    //------------------------------------------------------------------------//
    // VERIFY  VERIFY VERIFY VERIFY VERIFY VERIFY VERIFY VERIFY VERIFY VERIFY //
    //------------------------------------------------------------------------//
    //Verify current substate.
A(;
L #_emc_water_subs;
L "dbCONST".BLK.EMC2.SUBS.CHARGE;
==I;
);
    S     #sqSequencer.STEP.ActionVerified; //Action verified

    //------------------------------------------------------------------------//
    // Action done:                                                           //
    //------------------------------------------------------------------------//
    O     #sqSequencer.STEP.ActionVerified;
    O     #smc.NO_VERIFIC;       //No verification , bypass verification code
    S     #sqSequencer.STEP.ActionFinished;






    //============================= STEP FOOTER ==============================//
    // AUTOCODE   AUTOCODE   AUTOCODE   AUTOCODE   AUTOCODE   AUTOCODE   AUTO //
    // Get Ready after action finished:                                       //
    //------------------------------------------------------------------------//
    A     #sqSequencer.STEP.ActionFinished;
    JCN   k006;

    //------------------------------------------------------------------------//
    // Reset Action finished flag, ready for next step action:                //
    //------------------------------------------------------------------------//
    R     #sqSequencer.STEP.ActionVerified;
    R     #sqSequencer.STEP.ActionFinished;

    //------------------------------------------------------------------------//
    // If ALL actions are finished:                                           //
    //------------------------------------------------------------------------//
    SET   ;
    S     #sqSequencer.STEP.Finished;
    R     #sqSequencer.STEP.Active;
    S     #sqSequencer.STEP.Done[06];

    //------------------------------------------------------------------------//
    // End Step action(s):                                                    //
    //------------------------------------------------------------------------//
    JU    k006;

//----------------------------------------------------------------------------//
// Finished Step Action(s):                                                   //
//----------------------------------------------------------------------------//
k006: NOP   0;

    A     #sqStepTimerExpired;
    S     #sqSequencer.STEP.WithError[06]; // Step error flag
    S     #sqSequencer.Error_Fault;
    R     #sqStepTimer.IN;

NETWORK
TITLE =S006:STEP-006::Begin Transition
    //------------------------------------------------------------------------//
    // Begin the transition code:                                             //
    //------------------------------------------------------------------------//
    A006: NOP   0;
    R     #sqStepTimer.IN;






    //============================= TRAN HEADER ==============================//
    // AUTOCODE   AUTOCODE   AUTOCODE   AUTOCODE   AUTOCODE   AUTOCODE   AUTO //
    // Bypass transition if manual jump:                                      //
    //------------------------------------------------------------------------//
    A     #sqSequencer.STEP.Finished;
    A     #smc.TRN_AND_JUMP;     //Manual jump is set Transition as bypassed
    JCN   COMM;              //exit

NETWORK
TITLE =S006::STEP 006:TRAN 010: Charge WFI complete?
//----------------------------------------------------------------------------//
// TRAN   TRAN   TRAN   TRAN   TRAN   TRAN   TRAN   TRAN   TRAN   TRAN   TRAN //
// TRAN   TRAN   TRAN   TRAN   TRAN   TRAN   TRAN   TRAN   TRAN   TRAN   TRAN //
//----------------------------------------------------------------------------//
// Check if charging WFI is completed.
//----------------------------------------------------------------------------//
// CONDITION   CONDITION   CONDITION   CONDITION   CONDITION   CONDITION   CO //
// CONDITION   CONDITION   CONDITION   CONDITION   CONDITION   CONDITION   CO //
//----------------------------------------------------------------------------//
A(;
L   #_emc_water_state;
L   "dbCONST".BLK.STATE.COMPLETED;
==I;
);






    //============================= TRAN FOOTER ==============================//
    // Transition jump control:                                               //
    //------------------------------------------------------------------------//
    A     #sqSequencer.STEP.JumpCtrl;
    S     #sqSequencer.STEP.Jump;
    S     #sqSequencer.STEP.jumpDone[06];

NETWORK
TITLE =S006:t010::TRANS-v: EXIT TRANSITION AND READY THE NEXT STEP
    //------------------------------------------------------------------------//
    // Check the jump flag and jump to the next step if the transition        //
    // condition is true and has set the jump flag:                           //
    //------------------------------------------------------------------------//
    A     #sqSequencer.STEP.Jump;
    JCN   x010;

    R     #sqSequencer.STEP.Jump;
    R     #sqSequencer.STEP.Finished;

    L     07;     // Load next STEPNO to jump to if transition satisfied
    T     #sqSequencer.STEP.NumberNext; //Next Step07.

    JU    COMM;              // Transition satisfied, Exit, go to next step
x010: NOP   0;






NETWORK
TITLE =S006::STEP-006:EXIT TRANSITION:
    //========================== STEP TRANSFER ===============================//
    // Jump to the common step progression code:                              //
    //------------------------------------------------------------------------//
    JU    COMM;






NETWORK
TITLE =S007: STEP-07::UO_MX_MAKE : Reset command
    //================================ STEP HEADER ===========================//
    // STEP007 STEP007 STEP007 STEP007
    // AUTOCODE   AUTOCODE   AUTOCODE   AUTOCODE   AUTOCODE   AUTOCODE   AUTO //
    // STEP007 STEP007 STEP007 STEP007
    //------------------------------------------------------------------------//
    // Reset CHARGE command.
    // Log Mx vessel weight.
    //------------------------------------------------------------------------//
S007: NOP   0;

      SET;
      R     #sqSequencer.STEP.jumpDone[07];
      A     #sqSequencer.CMD.Pause; //If paused jump
      JC    COMM;

NETWORK
TITLE =S007:STEP-07:Begin Action

      A     #sqSequencer.STEP.Finished;
      JC    A007; // Exit Action code, Jump to A007 Transition code

      //----------------------------------------------------------------------//
      // Begin step Action:                                                   //
      //----------------------------------------------------------------------//
      A     #sqSequencer.STEP.Active;
      JC    L007; // Action number loaded, Jump to L007--Step Action List

      //----------------------------------------------------------------------//
      // Load Default/Initial Step action number:                             //
      //----------------------------------------------------------------------//
      S     #sqSequencer.STEP.Active;
      S     #sqStepTimer.IN;
      L     1; //First Action, Step must contain Minimum one action
      T     #sqSequencer.STEP.ActionNumber;

//----------------------------------------------------------------------------//
// Step action list.                                                          //
// aann=mini Action step number(aa) inside main step number(nn)               //
// First Action aa00, Second action ab00, Third ac00, etc.                    //
//----------------------------------------------------------------------------//
L007: NOP   0;

      L     #sqSequencer.STEP.ActionNumber;
      JL    r007; //Wrong Action number
      JU    _007; //Action error handling
       JU    aa07; //ACTION-01


//----------------------------------------------------------------------------//
// More step action in the list can be inserted here, upto ab is tested:      //
//----------------------------------------------------------------------------//
r007: NOP   0; //Wrong action number
      S     #sqSequencer.Error_Fault;
      JU    k007; //Exit
_007: NOP   0; // Action error handling
      JU    k007; // Exit






NETWORK
TITLE =S007:: STEP-007:: : ACTION CODE
    //================================ ACT HEADER ============================//
    // ACTION ACTION ACTION ACTION ACTION ACTION ACTION ACTION ACTION ACTION  //
    // AUTOCODE   AUTOCODE   AUTOCODE   AUTOCODE   AUTOCODE   AUTOCODE   AUTO //
    // ACTION ACTION ACTION ACTION ACTION ACTION ACTION ACTION ACTION ACTION  //
    //------------------------------------------------------------------------//
    // //Reset CHARGE command.
    aa07: NOP   0;

    //------------------------------------------------------------------------//
    // ACT ACT ACT ACT ACT ACT ACT ACT ACT ACT ACT ACT ACT ACT ACT ACT ACT    //
    //------------------------------------------------------------------------//
    L "dbCONST".BLK.CMD.STOP;
T #_emv_inlet_cmd;

// Reset flag.
SET;
R #_cmd_charge;

    //------------------------------------------------------------------------//
    // VERIFY  VERIFY VERIFY VERIFY VERIFY VERIFY VERIFY VERIFY VERIFY VERIFY //
    //------------------------------------------------------------------------//
    A "uncondJump";
    S     #sqSequencer.STEP.ActionVerified; //Action verified

    //------------------------------------------------------------------------//
    // Action done:                                                           //
    //------------------------------------------------------------------------//
    O     #sqSequencer.STEP.ActionVerified;
    O     #smc.NO_VERIFIC;       //No verification , bypass verification code
    S     #sqSequencer.STEP.ActionFinished;






    //============================= STEP FOOTER ==============================//
    // AUTOCODE   AUTOCODE   AUTOCODE   AUTOCODE   AUTOCODE   AUTOCODE   AUTO //
    // Get Ready after action finished:                                       //
    //------------------------------------------------------------------------//
    A     #sqSequencer.STEP.ActionFinished;
    JCN   k007;

    //------------------------------------------------------------------------//
    // Reset Action finished flag, ready for next step action:                //
    //------------------------------------------------------------------------//
    R     #sqSequencer.STEP.ActionVerified;
    R     #sqSequencer.STEP.ActionFinished;

    //------------------------------------------------------------------------//
    // If ALL actions are finished:                                           //
    //------------------------------------------------------------------------//
    SET   ;
    S     #sqSequencer.STEP.Finished;
    R     #sqSequencer.STEP.Active;
    S     #sqSequencer.STEP.Done[07];

    //------------------------------------------------------------------------//
    // End Step action(s):                                                    //
    //------------------------------------------------------------------------//
    JU    k007;

//----------------------------------------------------------------------------//
// Finished Step Action(s):                                                   //
//----------------------------------------------------------------------------//
k007: NOP   0;

    A     #sqStepTimerExpired;
    S     #sqSequencer.STEP.WithError[07]; // Step error flag
    S     #sqSequencer.Error_Fault;
    R     #sqStepTimer.IN;

NETWORK
TITLE =S007:STEP-007::Begin Transition
    //------------------------------------------------------------------------//
    // Begin the transition code:                                             //
    //------------------------------------------------------------------------//
    A007: NOP   0;
    R     #sqStepTimer.IN;






    //============================= TRAN HEADER ==============================//
    // AUTOCODE   AUTOCODE   AUTOCODE   AUTOCODE   AUTOCODE   AUTOCODE   AUTO //
    // Bypass transition if manual jump:                                      //
    //------------------------------------------------------------------------//
    A     #sqSequencer.STEP.Finished;
    A     #smc.TRN_AND_JUMP;     //Manual jump is set Transition as bypassed
    JCN   COMM;              //exit

NETWORK
TITLE =S007::STEP 007:TRAN 011: Sprayball inlet valves closed
//----------------------------------------------------------------------------//
// TRAN   TRAN   TRAN   TRAN   TRAN   TRAN   TRAN   TRAN   TRAN   TRAN   TRAN //
// TRAN   TRAN   TRAN   TRAN   TRAN   TRAN   TRAN   TRAN   TRAN   TRAN   TRAN //
//----------------------------------------------------------------------------//
// Jump if sprayball valves closed
//----------------------------------------------------------------------------//
// CONDITION   CONDITION   CONDITION   CONDITION   CONDITION   CONDITION   CO //
// CONDITION   CONDITION   CONDITION   CONDITION   CONDITION   CONDITION   CO //
//----------------------------------------------------------------------------//
A(;
L   #_emv_inlet_state;
L   "dbCONST".BLK.STATE.STOPPED;
==I;
);






    //============================= TRAN FOOTER ==============================//
    // Transition jump control:                                               //
    //------------------------------------------------------------------------//
    A     #sqSequencer.STEP.JumpCtrl;
    S     #sqSequencer.STEP.Jump;
    S     #sqSequencer.STEP.jumpDone[07];

NETWORK
TITLE =S007:t011::TRANS-v: EXIT TRANSITION AND READY THE NEXT STEP
    //------------------------------------------------------------------------//
    // Check the jump flag and jump to the next step if the transition        //
    // condition is true and has set the jump flag:                           //
    //------------------------------------------------------------------------//
    A     #sqSequencer.STEP.Jump;
    JCN   x011;

    R     #sqSequencer.STEP.Jump;
    R     #sqSequencer.STEP.Finished;

    L     03;     // Load next STEPNO to jump to if transition satisfied
    T     #sqSequencer.STEP.NumberNext; //Next Step03.

    JU    COMM;              // Transition satisfied, Exit, go to next step
x011: NOP   0;






NETWORK
TITLE =S007::STEP-007:EXIT TRANSITION:
    //========================== STEP TRANSFER ===============================//
    // Jump to the common step progression code:                              //
    //------------------------------------------------------------------------//
    JU    COMM;






NETWORK
TITLE =S008: STEP-08::UO_MX_MAKE : MIXING vessel contents
    //================================ STEP HEADER ===========================//
    // STEP008 STEP008 STEP008 STEP008
    // AUTOCODE   AUTOCODE   AUTOCODE   AUTOCODE   AUTOCODE   AUTOCODE   AUTO //
    // STEP008 STEP008 STEP008 STEP008
    //------------------------------------------------------------------------//
    // Set ema_vessel to substate MIX with pre-selected runtime and speed.
    //------------------------------------------------------------------------//
S008: NOP   0;

      SET;
      R     #sqSequencer.STEP.jumpDone[08];
      A     #sqSequencer.CMD.Pause; //If paused jump
      JC    COMM;

NETWORK
TITLE =S008:STEP-08:Begin Action

      A     #sqSequencer.STEP.Finished;
      JC    A008; // Exit Action code, Jump to A008 Transition code

      //----------------------------------------------------------------------//
      // Begin step Action:                                                   //
      //----------------------------------------------------------------------//
      A     #sqSequencer.STEP.Active;
      JC    L008; // Action number loaded, Jump to L008--Step Action List

      //----------------------------------------------------------------------//
      // Load Default/Initial Step action number:                             //
      //----------------------------------------------------------------------//
      S     #sqSequencer.STEP.Active;
      S     #sqStepTimer.IN;
      L     1; //First Action, Step must contain Minimum one action
      T     #sqSequencer.STEP.ActionNumber;

//----------------------------------------------------------------------------//
// Step action list.                                                          //
// aann=mini Action step number(aa) inside main step number(nn)               //
// First Action aa00, Second action ab00, Third ac00, etc.                    //
//----------------------------------------------------------------------------//
L008: NOP   0;

      L     #sqSequencer.STEP.ActionNumber;
      JL    r008; //Wrong Action number
      JU    _008; //Action error handling
       JU    aa08; //ACTION-01
JU    ab08; //ACTION-02


//----------------------------------------------------------------------------//
// More step action in the list can be inserted here, upto ab is tested:      //
//----------------------------------------------------------------------------//
r008: NOP   0; //Wrong action number
      S     #sqSequencer.Error_Fault;
      JU    k008; //Exit
_008: NOP   0; // Action error handling
      JU    k008; // Exit






NETWORK
TITLE =S008:: STEP-008:: : ACTION CODE
    //================================ ACT HEADER ============================//
    // ACTION ACTION ACTION ACTION ACTION ACTION ACTION ACTION ACTION ACTION  //
    // AUTOCODE   AUTOCODE   AUTOCODE   AUTOCODE   AUTOCODE   AUTOCODE   AUTO //
    // ACTION ACTION ACTION ACTION ACTION ACTION ACTION ACTION ACTION ACTION  //
    //------------------------------------------------------------------------//
    // //Set substate to safe state and stop ema_vessel.
    aa08: NOP   0;

    //------------------------------------------------------------------------//
    // ACT ACT ACT ACT ACT ACT ACT ACT ACT ACT ACT ACT ACT ACT ACT ACT ACT    //
    //------------------------------------------------------------------------//
    L "dbCONST".BLK.CMD.STOP;
T  #_ema_vessel_cmd;

    //------------------------------------------------------------------------//
    // VERIFY  VERIFY VERIFY VERIFY VERIFY VERIFY VERIFY VERIFY VERIFY VERIFY //
    //------------------------------------------------------------------------//
    //Verify ema_vessel stopped status.
A(;
L #_ema_vessel_state;
L "dbCONST".BLK.STATE.STOPPED;
==I;
);
    S     #sqSequencer.STEP.ActionVerified; //Action verified

    //------------------------------------------------------------------------//
    // Action done:                                                           //
    //------------------------------------------------------------------------//
    O     #sqSequencer.STEP.ActionVerified;
    O     #smc.NO_VERIFIC;       //No verification , bypass verification code
    S     #sqSequencer.STEP.ActionFinished;






    //============================= ACT FOOTER ===============================//
    // AUTOCODE   AUTOCODE   AUTOCODE   AUTOCODE   AUTOCODE   AUTOCODE   AUTO //
    // Get Ready after action finished:                                       //
    //------------------------------------------------------------------------//
    A     #sqSequencer.STEP.ActionFinished;
    JCN   k008;

    //------------------------------------------------------------------------//
    // Reset Action finished flag, ready for next step action:                //
    //------------------------------------------------------------------------//
    R     #sqSequencer.STEP.ActionVerified;
    R     #sqSequencer.STEP.ActionFinished;

    //------------------------------------------------------------------------//
    // Load Next Step Action number:                                          //
    //------------------------------------------------------------------------//
    L     02; //Load next Action
    T     #sqSequencer.STEP.ActionNumber;






NETWORK
TITLE =S008:: STEP-008:: : ACTION CODE
    //================================ ACT HEADER ============================//
    // ACTION ACTION ACTION ACTION ACTION ACTION ACTION ACTION ACTION ACTION  //
    // AUTOCODE   AUTOCODE   AUTOCODE   AUTOCODE   AUTOCODE   AUTOCODE   AUTO //
    // ACTION ACTION ACTION ACTION ACTION ACTION ACTION ACTION ACTION ACTION  //
    //------------------------------------------------------------------------//
    // //Set ema_vessel to substate MIX with pre-selected timeout and speed.
    ab08: NOP   0;

    //------------------------------------------------------------------------//
    // ACT ACT ACT ACT ACT ACT ACT ACT ACT ACT ACT ACT ACT ACT ACT ACT ACT    //
    //------------------------------------------------------------------------//
    //Transfer input parameter from HMI to EM
//Load Agitator speed setpoint.
L #_fp_speed_setpoint;
T #_ema_vessel_setpoint;
//Load Agitator runtime.
L #_fp_time_make_agit;
L 1000;
*I;
T #_ema_vessel_runtime;

// Start Agitator
L "dbCONST".BLK.EMA1.SUBS.MIX;
T #_ema_vessel_subs;
L "dbCONST".BLK.CMD.START;
T #_ema_vessel_cmd;

    //------------------------------------------------------------------------//
    // VERIFY  VERIFY VERIFY VERIFY VERIFY VERIFY VERIFY VERIFY VERIFY VERIFY //
    //------------------------------------------------------------------------//
    //Substate changed to Mix.
A(;
L #_ema_vessel_subs;
L "dbCONST".BLK.EMA1.SUBS.MIX;
==I;
);
    S     #sqSequencer.STEP.ActionVerified; //Action verified

    //------------------------------------------------------------------------//
    // Action done:                                                           //
    //------------------------------------------------------------------------//
    O     #sqSequencer.STEP.ActionVerified;
    O     #smc.NO_VERIFIC;       //No verification , bypass verification code
    S     #sqSequencer.STEP.ActionFinished;






    //============================= STEP FOOTER ==============================//
    // AUTOCODE   AUTOCODE   AUTOCODE   AUTOCODE   AUTOCODE   AUTOCODE   AUTO //
    // Get Ready after action finished:                                       //
    //------------------------------------------------------------------------//
    A     #sqSequencer.STEP.ActionFinished;
    JCN   k008;

    //------------------------------------------------------------------------//
    // Reset Action finished flag, ready for next step action:                //
    //------------------------------------------------------------------------//
    R     #sqSequencer.STEP.ActionVerified;
    R     #sqSequencer.STEP.ActionFinished;

    //------------------------------------------------------------------------//
    // If ALL actions are finished:                                           //
    //------------------------------------------------------------------------//
    SET   ;
    S     #sqSequencer.STEP.Finished;
    R     #sqSequencer.STEP.Active;
    S     #sqSequencer.STEP.Done[08];

    //------------------------------------------------------------------------//
    // End Step action(s):                                                    //
    //------------------------------------------------------------------------//
    JU    k008;

//----------------------------------------------------------------------------//
// Finished Step Action(s):                                                   //
//----------------------------------------------------------------------------//
k008: NOP   0;

    A     #sqStepTimerExpired;
    S     #sqSequencer.STEP.WithError[08]; // Step error flag
    S     #sqSequencer.Error_Fault;
    R     #sqStepTimer.IN;

NETWORK
TITLE =S008:STEP-008::Begin Transition
    //------------------------------------------------------------------------//
    // Begin the transition code:                                             //
    //------------------------------------------------------------------------//
    A008: NOP   0;
    R     #sqStepTimer.IN;






    //============================= TRAN HEADER ==============================//
    // AUTOCODE   AUTOCODE   AUTOCODE   AUTOCODE   AUTOCODE   AUTOCODE   AUTO //
    // Bypass transition if manual jump:                                      //
    //------------------------------------------------------------------------//
    A     #sqSequencer.STEP.Finished;
    A     #smc.TRN_AND_JUMP;     //Manual jump is set Transition as bypassed
    JCN   COMM;              //exit

NETWORK
TITLE =S008::STEP 008:TRAN 012: Mixing complete?
//----------------------------------------------------------------------------//
// TRAN   TRAN   TRAN   TRAN   TRAN   TRAN   TRAN   TRAN   TRAN   TRAN   TRAN //
// TRAN   TRAN   TRAN   TRAN   TRAN   TRAN   TRAN   TRAN   TRAN   TRAN   TRAN //
//----------------------------------------------------------------------------//
// Check if Mixing is completed.
//----------------------------------------------------------------------------//
// CONDITION   CONDITION   CONDITION   CONDITION   CONDITION   CONDITION   CO //
// CONDITION   CONDITION   CONDITION   CONDITION   CONDITION   CONDITION   CO //
//----------------------------------------------------------------------------//
A(;
L   #_ema_vessel_state;
L   "dbCONST".BLK.STATE.COMPLETED;
==I;
);






    //============================= TRAN FOOTER ==============================//
    // Transition jump control:                                               //
    //------------------------------------------------------------------------//
    A     #sqSequencer.STEP.JumpCtrl;
    S     #sqSequencer.STEP.Jump;
    S     #sqSequencer.STEP.jumpDone[08];

NETWORK
TITLE =S008:t012::TRANS-v: EXIT TRANSITION AND READY THE NEXT STEP
    //------------------------------------------------------------------------//
    // Check the jump flag and jump to the next step if the transition        //
    // condition is true and has set the jump flag:                           //
    //------------------------------------------------------------------------//
    A     #sqSequencer.STEP.Jump;
    JCN   x012;

    R     #sqSequencer.STEP.Jump;
    R     #sqSequencer.STEP.Finished;

    L     09;     // Load next STEPNO to jump to if transition satisfied
    T     #sqSequencer.STEP.NumberNext; //Next Step09.

    JU    COMM;              // Transition satisfied, Exit, go to next step
x012: NOP   0;






NETWORK
TITLE =S008::STEP-008:EXIT TRANSITION:
    //========================== STEP TRANSFER ===============================//
    // Jump to the common step progression code:                              //
    //------------------------------------------------------------------------//
    JU    COMM;






NETWORK
TITLE =S009: STEP-09::UO_MX_MAKE : Reset MIX command.
    //================================ STEP HEADER ===========================//
    // STEP009 STEP009 STEP009 STEP009
    // AUTOCODE   AUTOCODE   AUTOCODE   AUTOCODE   AUTOCODE   AUTOCODE   AUTO //
    // STEP009 STEP009 STEP009 STEP009
    //------------------------------------------------------------------------//
    // Reset MIX command.
    //------------------------------------------------------------------------//
S009: NOP   0;

      SET;
      R     #sqSequencer.STEP.jumpDone[09];
      A     #sqSequencer.CMD.Pause; //If paused jump
      JC    COMM;

NETWORK
TITLE =S009:STEP-09:Begin Action

      A     #sqSequencer.STEP.Finished;
      JC    A009; // Exit Action code, Jump to A009 Transition code

      //----------------------------------------------------------------------//
      // Begin step Action:                                                   //
      //----------------------------------------------------------------------//
      A     #sqSequencer.STEP.Active;
      JC    L009; // Action number loaded, Jump to L009--Step Action List

      //----------------------------------------------------------------------//
      // Load Default/Initial Step action number:                             //
      //----------------------------------------------------------------------//
      S     #sqSequencer.STEP.Active;
      S     #sqStepTimer.IN;
      L     1; //First Action, Step must contain Minimum one action
      T     #sqSequencer.STEP.ActionNumber;

//----------------------------------------------------------------------------//
// Step action list.                                                          //
// aann=mini Action step number(aa) inside main step number(nn)               //
// First Action aa00, Second action ab00, Third ac00, etc.                    //
//----------------------------------------------------------------------------//
L009: NOP   0;

      L     #sqSequencer.STEP.ActionNumber;
      JL    r009; //Wrong Action number
      JU    _009; //Action error handling
       JU    aa09; //ACTION-01


//----------------------------------------------------------------------------//
// More step action in the list can be inserted here, upto ab is tested:      //
//----------------------------------------------------------------------------//
r009: NOP   0; //Wrong action number
      S     #sqSequencer.Error_Fault;
      JU    k009; //Exit
_009: NOP   0; // Action error handling
      JU    k009; // Exit






NETWORK
TITLE =S009:: STEP-009:: : ACTION CODE
    //================================ ACT HEADER ============================//
    // ACTION ACTION ACTION ACTION ACTION ACTION ACTION ACTION ACTION ACTION  //
    // AUTOCODE   AUTOCODE   AUTOCODE   AUTOCODE   AUTOCODE   AUTOCODE   AUTO //
    // ACTION ACTION ACTION ACTION ACTION ACTION ACTION ACTION ACTION ACTION  //
    //------------------------------------------------------------------------//
    // //Reset CHARGE command.
    aa09: NOP   0;

    //------------------------------------------------------------------------//
    // ACT ACT ACT ACT ACT ACT ACT ACT ACT ACT ACT ACT ACT ACT ACT ACT ACT    //
    //------------------------------------------------------------------------//
    // Reset flag.
SET;
R #_cmd_mix;

    //------------------------------------------------------------------------//
    // VERIFY  VERIFY VERIFY VERIFY VERIFY VERIFY VERIFY VERIFY VERIFY VERIFY //
    //------------------------------------------------------------------------//
    A "uncondJump";
    S     #sqSequencer.STEP.ActionVerified; //Action verified

    //------------------------------------------------------------------------//
    // Action done:                                                           //
    //------------------------------------------------------------------------//
    O     #sqSequencer.STEP.ActionVerified;
    O     #smc.NO_VERIFIC;       //No verification , bypass verification code
    S     #sqSequencer.STEP.ActionFinished;






    //============================= STEP FOOTER ==============================//
    // AUTOCODE   AUTOCODE   AUTOCODE   AUTOCODE   AUTOCODE   AUTOCODE   AUTO //
    // Get Ready after action finished:                                       //
    //------------------------------------------------------------------------//
    A     #sqSequencer.STEP.ActionFinished;
    JCN   k009;

    //------------------------------------------------------------------------//
    // Reset Action finished flag, ready for next step action:                //
    //------------------------------------------------------------------------//
    R     #sqSequencer.STEP.ActionVerified;
    R     #sqSequencer.STEP.ActionFinished;

    //------------------------------------------------------------------------//
    // If ALL actions are finished:                                           //
    //------------------------------------------------------------------------//
    SET   ;
    S     #sqSequencer.STEP.Finished;
    R     #sqSequencer.STEP.Active;
    S     #sqSequencer.STEP.Done[09];

    //------------------------------------------------------------------------//
    // End Step action(s):                                                    //
    //------------------------------------------------------------------------//
    JU    k009;

//----------------------------------------------------------------------------//
// Finished Step Action(s):                                                   //
//----------------------------------------------------------------------------//
k009: NOP   0;

    A     #sqStepTimerExpired;
    S     #sqSequencer.STEP.WithError[09]; // Step error flag
    S     #sqSequencer.Error_Fault;
    R     #sqStepTimer.IN;

NETWORK
TITLE =S009:STEP-009::Begin Transition
    //------------------------------------------------------------------------//
    // Begin the transition code:                                             //
    //------------------------------------------------------------------------//
    A009: NOP   0;
    R     #sqStepTimer.IN;






    //============================= TRAN HEADER ==============================//
    // AUTOCODE   AUTOCODE   AUTOCODE   AUTOCODE   AUTOCODE   AUTOCODE   AUTO //
    // Bypass transition if manual jump:                                      //
    //------------------------------------------------------------------------//
    A     #sqSequencer.STEP.Finished;
    A     #smc.TRN_AND_JUMP;     //Manual jump is set Transition as bypassed
    JCN   COMM;              //exit

NETWORK
TITLE =S009::STEP 009:TRAN 013: Empty Transition
//----------------------------------------------------------------------------//
// TRAN   TRAN   TRAN   TRAN   TRAN   TRAN   TRAN   TRAN   TRAN   TRAN   TRAN //
// TRAN   TRAN   TRAN   TRAN   TRAN   TRAN   TRAN   TRAN   TRAN   TRAN   TRAN //
//----------------------------------------------------------------------------//
// Jump
//----------------------------------------------------------------------------//
// CONDITION   CONDITION   CONDITION   CONDITION   CONDITION   CONDITION   CO //
// CONDITION   CONDITION   CONDITION   CONDITION   CONDITION   CONDITION   CO //
//----------------------------------------------------------------------------//
A "uncondJump";






    //============================= TRAN FOOTER ==============================//
    // Transition jump control:                                               //
    //------------------------------------------------------------------------//
    A     #sqSequencer.STEP.JumpCtrl;
    S     #sqSequencer.STEP.Jump;
    S     #sqSequencer.STEP.jumpDone[09];

NETWORK
TITLE =S009:t013::TRANS-v: EXIT TRANSITION AND READY THE NEXT STEP
    //------------------------------------------------------------------------//
    // Check the jump flag and jump to the next step if the transition        //
    // condition is true and has set the jump flag:                           //
    //------------------------------------------------------------------------//
    A     #sqSequencer.STEP.Jump;
    JCN   x013;

    R     #sqSequencer.STEP.Jump;
    R     #sqSequencer.STEP.Finished;

    L     03;     // Load next STEPNO to jump to if transition satisfied
    T     #sqSequencer.STEP.NumberNext; //Next Step03.

    JU    COMM;              // Transition satisfied, Exit, go to next step
x013: NOP   0;






NETWORK
TITLE =S009::STEP-009:EXIT TRANSITION:
    //========================== STEP TRANSFER ===============================//
    // Jump to the common step progression code:                              //
    //------------------------------------------------------------------------//
    JU    COMM;






NETWORK
TITLE =S010: STEP-10::UO_MX_MAKE : Disabling manway alarm
    //================================ STEP HEADER ===========================//
    // STEP010 STEP010 STEP010 STEP010
    // AUTOCODE   AUTOCODE   AUTOCODE   AUTOCODE   AUTOCODE   AUTOCODE   AUTO //
    // STEP010 STEP010 STEP010 STEP010
    //------------------------------------------------------------------------//
    // Disable Mx Low and LowLow Pressure Alarm.
    // Disable Mx manway alarm.
    //------------------------------------------------------------------------//
S010: NOP   0;

      SET;
      R     #sqSequencer.STEP.jumpDone[10];
      A     #sqSequencer.CMD.Pause; //If paused jump
      JC    COMM;

NETWORK
TITLE =S010:STEP-10:Begin Action

      A     #sqSequencer.STEP.Finished;
      JC    A010; // Exit Action code, Jump to A010 Transition code

      //----------------------------------------------------------------------//
      // Begin step Action:                                                   //
      //----------------------------------------------------------------------//
      A     #sqSequencer.STEP.Active;
      JC    L010; // Action number loaded, Jump to L010--Step Action List

      //----------------------------------------------------------------------//
      // Load Default/Initial Step action number:                             //
      //----------------------------------------------------------------------//
      S     #sqSequencer.STEP.Active;
      S     #sqStepTimer.IN;
      L     1; //First Action, Step must contain Minimum one action
      T     #sqSequencer.STEP.ActionNumber;

//----------------------------------------------------------------------------//
// Step action list.                                                          //
// aann=mini Action step number(aa) inside main step number(nn)               //
// First Action aa00, Second action ab00, Third ac00, etc.                    //
//----------------------------------------------------------------------------//
L010: NOP   0;

      L     #sqSequencer.STEP.ActionNumber;
      JL    r010; //Wrong Action number
      JU    _010; //Action error handling
       JU    aa10; //ACTION-01
JU    ab10; //ACTION-02


//----------------------------------------------------------------------------//
// More step action in the list can be inserted here, upto ab is tested:      //
//----------------------------------------------------------------------------//
r010: NOP   0; //Wrong action number
      S     #sqSequencer.Error_Fault;
      JU    k010; //Exit
_010: NOP   0; // Action error handling
      JU    k010; // Exit






NETWORK
TITLE =S010:: STEP-010:: : ACTION CODE
    //================================ ACT HEADER ============================//
    // ACTION ACTION ACTION ACTION ACTION ACTION ACTION ACTION ACTION ACTION  //
    // AUTOCODE   AUTOCODE   AUTOCODE   AUTOCODE   AUTOCODE   AUTOCODE   AUTO //
    // ACTION ACTION ACTION ACTION ACTION ACTION ACTION ACTION ACTION ACTION  //
    //------------------------------------------------------------------------//
    // //Close LPCA valve
    aa10: NOP   0;

    //------------------------------------------------------------------------//
    // ACT ACT ACT ACT ACT ACT ACT ACT ACT ACT ACT ACT ACT ACT ACT ACT ACT    //
    //------------------------------------------------------------------------//
    //Set substate to safe state and stop emc_gas.
L "dbCONST".BLK.CMD.STOP;
T  #_emc_gas_cmd;

    //------------------------------------------------------------------------//
    // VERIFY  VERIFY VERIFY VERIFY VERIFY VERIFY VERIFY VERIFY VERIFY VERIFY //
    //------------------------------------------------------------------------//
    //Verify emc_gas stopped.
A(;
L #_emc_gas_state;
L "dbCONST".BLK.STATE.STOPPED;
==I;
);
    S     #sqSequencer.STEP.ActionVerified; //Action verified

    //------------------------------------------------------------------------//
    // Action done:                                                           //
    //------------------------------------------------------------------------//
    O     #sqSequencer.STEP.ActionVerified;
    O     #smc.NO_VERIFIC;       //No verification , bypass verification code
    S     #sqSequencer.STEP.ActionFinished;






    //============================= ACT FOOTER ===============================//
    // AUTOCODE   AUTOCODE   AUTOCODE   AUTOCODE   AUTOCODE   AUTOCODE   AUTO //
    // Get Ready after action finished:                                       //
    //------------------------------------------------------------------------//
    A     #sqSequencer.STEP.ActionFinished;
    JCN   k010;

    //------------------------------------------------------------------------//
    // Reset Action finished flag, ready for next step action:                //
    //------------------------------------------------------------------------//
    R     #sqSequencer.STEP.ActionVerified;
    R     #sqSequencer.STEP.ActionFinished;

    //------------------------------------------------------------------------//
    // Load Next Step Action number:                                          //
    //------------------------------------------------------------------------//
    L     02; //Load next Action
    T     #sqSequencer.STEP.ActionNumber;






NETWORK
TITLE =S010:: STEP-010:: : ACTION CODE
    //================================ ACT HEADER ============================//
    // ACTION ACTION ACTION ACTION ACTION ACTION ACTION ACTION ACTION ACTION  //
    // AUTOCODE   AUTOCODE   AUTOCODE   AUTOCODE   AUTOCODE   AUTOCODE   AUTO //
    // ACTION ACTION ACTION ACTION ACTION ACTION ACTION ACTION ACTION ACTION  //
    //------------------------------------------------------------------------//
    // //Disable Mx Low and LowLow Pressure Alarm.
    // //Disable Mx manway alarm and prompt operator to confirm when MANWAY disabling finished.
    ab10: NOP   0;

    //------------------------------------------------------------------------//
    // ACT ACT ACT ACT ACT ACT ACT ACT ACT ACT ACT ACT ACT ACT ACT ACT ACT    //
    //------------------------------------------------------------------------//
    //Set emv_vessel to substate MANWAY and start it to disable Manway alarm.
L "dbCONST".BLK.EMV1.SUBS.MANWAY;
T #_emv_vessel_subs;
L "dbCONST".BLK.CMD.START;
T #_emv_vessel_cmd;


SET;
S #_prompt_manway_complete;

    //------------------------------------------------------------------------//
    // VERIFY  VERIFY VERIFY VERIFY VERIFY VERIFY VERIFY VERIFY VERIFY VERIFY //
    //------------------------------------------------------------------------//
    //Verify emv_vessel changed to substate MANWAY.
A(;
L #_emv_vessel_subs;
L "dbCONST".BLK.EMV1.SUBS.MANWAY;
==I;
);
    S     #sqSequencer.STEP.ActionVerified; //Action verified

    //------------------------------------------------------------------------//
    // Action done:                                                           //
    //------------------------------------------------------------------------//
    O     #sqSequencer.STEP.ActionVerified;
    O     #smc.NO_VERIFIC;       //No verification , bypass verification code
    S     #sqSequencer.STEP.ActionFinished;






    //============================= STEP FOOTER ==============================//
    // AUTOCODE   AUTOCODE   AUTOCODE   AUTOCODE   AUTOCODE   AUTOCODE   AUTO //
    // Get Ready after action finished:                                       //
    //------------------------------------------------------------------------//
    A     #sqSequencer.STEP.ActionFinished;
    JCN   k010;

    //------------------------------------------------------------------------//
    // Reset Action finished flag, ready for next step action:                //
    //------------------------------------------------------------------------//
    R     #sqSequencer.STEP.ActionVerified;
    R     #sqSequencer.STEP.ActionFinished;

    //------------------------------------------------------------------------//
    // If ALL actions are finished:                                           //
    //------------------------------------------------------------------------//
    SET   ;
    S     #sqSequencer.STEP.Finished;
    R     #sqSequencer.STEP.Active;
    S     #sqSequencer.STEP.Done[10];

    //------------------------------------------------------------------------//
    // End Step action(s):                                                    //
    //------------------------------------------------------------------------//
    JU    k010;

//----------------------------------------------------------------------------//
// Finished Step Action(s):                                                   //
//----------------------------------------------------------------------------//
k010: NOP   0;

    A     #sqStepTimerExpired;
    S     #sqSequencer.STEP.WithError[10]; // Step error flag
    S     #sqSequencer.Error_Fault;
    R     #sqStepTimer.IN;

NETWORK
TITLE =S010:STEP-010::Begin Transition
    //------------------------------------------------------------------------//
    // Begin the transition code:                                             //
    //------------------------------------------------------------------------//
    A010: NOP   0;
    R     #sqStepTimer.IN;






    //============================= TRAN HEADER ==============================//
    // AUTOCODE   AUTOCODE   AUTOCODE   AUTOCODE   AUTOCODE   AUTOCODE   AUTO //
    // Bypass transition if manual jump:                                      //
    //------------------------------------------------------------------------//
    A     #sqSequencer.STEP.Finished;
    A     #smc.TRN_AND_JUMP;     //Manual jump is set Transition as bypassed
    JCN   COMM;              //exit

NETWORK
TITLE =S010::STEP 010:TRAN 014: Complete with MANWAY charges?
//----------------------------------------------------------------------------//
// TRAN   TRAN   TRAN   TRAN   TRAN   TRAN   TRAN   TRAN   TRAN   TRAN   TRAN //
// TRAN   TRAN   TRAN   TRAN   TRAN   TRAN   TRAN   TRAN   TRAN   TRAN   TRAN //
//----------------------------------------------------------------------------//
// Operator confirm charges via MANWAY are completed.
//----------------------------------------------------------------------------//
// CONDITION   CONDITION   CONDITION   CONDITION   CONDITION   CONDITION   CO //
// CONDITION   CONDITION   CONDITION   CONDITION   CONDITION   CONDITION   CO //
//----------------------------------------------------------------------------//
A #_prompt_manway_complete_confirm_yes;






    //============================= TRAN FOOTER ==============================//
    // Transition jump control:                                               //
    //------------------------------------------------------------------------//
    A     #sqSequencer.STEP.JumpCtrl;
    S     #sqSequencer.STEP.Jump;
    S     #sqSequencer.STEP.jumpDone[10];

NETWORK
TITLE =S010:t014::TRANS-v: EXIT TRANSITION AND READY THE NEXT STEP
    //------------------------------------------------------------------------//
    // Check the jump flag and jump to the next step if the transition        //
    // condition is true and has set the jump flag:                           //
    //------------------------------------------------------------------------//
    A     #sqSequencer.STEP.Jump;
    JCN   x014;

    R     #sqSequencer.STEP.Jump;
    R     #sqSequencer.STEP.Finished;

    L     11;     // Load next STEPNO to jump to if transition satisfied
    T     #sqSequencer.STEP.NumberNext; //Next Step11.

    JU    COMM;              // Transition satisfied, Exit, go to next step
x014: NOP   0;






NETWORK
TITLE =S010::STEP-010:EXIT TRANSITION:
    //========================== STEP TRANSFER ===============================//
    // Jump to the common step progression code:                              //
    //------------------------------------------------------------------------//
    JU    COMM;






NETWORK
TITLE =S011: STEP-11::UO_MX_MAKE : Reset command
    //================================ STEP HEADER ===========================//
    // STEP011 STEP011 STEP011 STEP011
    // AUTOCODE   AUTOCODE   AUTOCODE   AUTOCODE   AUTOCODE   AUTOCODE   AUTO //
    // STEP011 STEP011 STEP011 STEP011
    //------------------------------------------------------------------------//
    // Enable MANWAY alarm and reset MANWAY command.
    //------------------------------------------------------------------------//
S011: NOP   0;

      SET;
      R     #sqSequencer.STEP.jumpDone[11];
      A     #sqSequencer.CMD.Pause; //If paused jump
      JC    COMM;

NETWORK
TITLE =S011:STEP-11:Begin Action

      A     #sqSequencer.STEP.Finished;
      JC    A011; // Exit Action code, Jump to A011 Transition code

      //----------------------------------------------------------------------//
      // Begin step Action:                                                   //
      //----------------------------------------------------------------------//
      A     #sqSequencer.STEP.Active;
      JC    L011; // Action number loaded, Jump to L011--Step Action List

      //----------------------------------------------------------------------//
      // Load Default/Initial Step action number:                             //
      //----------------------------------------------------------------------//
      S     #sqSequencer.STEP.Active;
      S     #sqStepTimer.IN;
      L     1; //First Action, Step must contain Minimum one action
      T     #sqSequencer.STEP.ActionNumber;

//----------------------------------------------------------------------------//
// Step action list.                                                          //
// aann=mini Action step number(aa) inside main step number(nn)               //
// First Action aa00, Second action ab00, Third ac00, etc.                    //
//----------------------------------------------------------------------------//
L011: NOP   0;

      L     #sqSequencer.STEP.ActionNumber;
      JL    r011; //Wrong Action number
      JU    _011; //Action error handling
       JU    aa11; //ACTION-01


//----------------------------------------------------------------------------//
// More step action in the list can be inserted here, upto ab is tested:      //
//----------------------------------------------------------------------------//
r011: NOP   0; //Wrong action number
      S     #sqSequencer.Error_Fault;
      JU    k011; //Exit
_011: NOP   0; // Action error handling
      JU    k011; // Exit






NETWORK
TITLE =S011:: STEP-011:: : ACTION CODE
    //================================ ACT HEADER ============================//
    // ACTION ACTION ACTION ACTION ACTION ACTION ACTION ACTION ACTION ACTION  //
    // AUTOCODE   AUTOCODE   AUTOCODE   AUTOCODE   AUTOCODE   AUTOCODE   AUTO //
    // ACTION ACTION ACTION ACTION ACTION ACTION ACTION ACTION ACTION ACTION  //
    //------------------------------------------------------------------------//
    // //Reset MANWAY command.
    aa11: NOP   0;

    //------------------------------------------------------------------------//
    // ACT ACT ACT ACT ACT ACT ACT ACT ACT ACT ACT ACT ACT ACT ACT ACT ACT    //
    //------------------------------------------------------------------------//
    T #_emv_vessel_subs;
L "dbCONST".BLK.CMD.STOP;
T #_emv_vessel_cmd;

// Enable LPCA control.
L #_r_pres_lpca_make;
T #_emc_gas_setpoint;
L "dbCONST".SEL.GAS.LPCA;
T #_emc_gas_medium_gas;
L "dbCONST".BLK.EMC1.SUBS.PRESSURE;
T #_emc_gas_subs;
L "dbCONST".BLK.CMD.START;
T #_emc_gas_cmd;

// Reset flags
SET;
R #_cmd_manway;
R #_prompt_manway_complete_confirm_yes;

    //------------------------------------------------------------------------//
    // VERIFY  VERIFY VERIFY VERIFY VERIFY VERIFY VERIFY VERIFY VERIFY VERIFY //
    //------------------------------------------------------------------------//
    A(;
L #_emc_gas_subs;
L "dbCONST".BLK.EMC1.SUBS.PRESSURE;
==I;
);
    S     #sqSequencer.STEP.ActionVerified; //Action verified

    //------------------------------------------------------------------------//
    // Action done:                                                           //
    //------------------------------------------------------------------------//
    O     #sqSequencer.STEP.ActionVerified;
    O     #smc.NO_VERIFIC;       //No verification , bypass verification code
    S     #sqSequencer.STEP.ActionFinished;






    //============================= STEP FOOTER ==============================//
    // AUTOCODE   AUTOCODE   AUTOCODE   AUTOCODE   AUTOCODE   AUTOCODE   AUTO //
    // Get Ready after action finished:                                       //
    //------------------------------------------------------------------------//
    A     #sqSequencer.STEP.ActionFinished;
    JCN   k011;

    //------------------------------------------------------------------------//
    // Reset Action finished flag, ready for next step action:                //
    //------------------------------------------------------------------------//
    R     #sqSequencer.STEP.ActionVerified;
    R     #sqSequencer.STEP.ActionFinished;

    //------------------------------------------------------------------------//
    // If ALL actions are finished:                                           //
    //------------------------------------------------------------------------//
    SET   ;
    S     #sqSequencer.STEP.Finished;
    R     #sqSequencer.STEP.Active;
    S     #sqSequencer.STEP.Done[11];

    //------------------------------------------------------------------------//
    // End Step action(s):                                                    //
    //------------------------------------------------------------------------//
    JU    k011;

//----------------------------------------------------------------------------//
// Finished Step Action(s):                                                   //
//----------------------------------------------------------------------------//
k011: NOP   0;

    A     #sqStepTimerExpired;
    S     #sqSequencer.STEP.WithError[11]; // Step error flag
    S     #sqSequencer.Error_Fault;
    R     #sqStepTimer.IN;

NETWORK
TITLE =S011:STEP-011::Begin Transition
    //------------------------------------------------------------------------//
    // Begin the transition code:                                             //
    //------------------------------------------------------------------------//
    A011: NOP   0;
    R     #sqStepTimer.IN;






    //============================= TRAN HEADER ==============================//
    // AUTOCODE   AUTOCODE   AUTOCODE   AUTOCODE   AUTOCODE   AUTOCODE   AUTO //
    // Bypass transition if manual jump:                                      //
    //------------------------------------------------------------------------//
    A     #sqSequencer.STEP.Finished;
    A     #smc.TRN_AND_JUMP;     //Manual jump is set Transition as bypassed
    JCN   COMM;              //exit

NETWORK
TITLE =S011::STEP 011:TRAN 015: Empty Transition
//----------------------------------------------------------------------------//
// TRAN   TRAN   TRAN   TRAN   TRAN   TRAN   TRAN   TRAN   TRAN   TRAN   TRAN //
// TRAN   TRAN   TRAN   TRAN   TRAN   TRAN   TRAN   TRAN   TRAN   TRAN   TRAN //
//----------------------------------------------------------------------------//
// Jump
//----------------------------------------------------------------------------//
// CONDITION   CONDITION   CONDITION   CONDITION   CONDITION   CONDITION   CO //
// CONDITION   CONDITION   CONDITION   CONDITION   CONDITION   CONDITION   CO //
//----------------------------------------------------------------------------//
A "uncondJump";






    //============================= TRAN FOOTER ==============================//
    // Transition jump control:                                               //
    //------------------------------------------------------------------------//
    A     #sqSequencer.STEP.JumpCtrl;
    S     #sqSequencer.STEP.Jump;
    S     #sqSequencer.STEP.jumpDone[11];

NETWORK
TITLE =S011:t015::TRANS-v: EXIT TRANSITION AND READY THE NEXT STEP
    //------------------------------------------------------------------------//
    // Check the jump flag and jump to the next step if the transition        //
    // condition is true and has set the jump flag:                           //
    //------------------------------------------------------------------------//
    A     #sqSequencer.STEP.Jump;
    JCN   x015;

    R     #sqSequencer.STEP.Jump;
    R     #sqSequencer.STEP.Finished;

    L     03;     // Load next STEPNO to jump to if transition satisfied
    T     #sqSequencer.STEP.NumberNext; //Next Step03.

    JU    COMM;              // Transition satisfied, Exit, go to next step
x015: NOP   0;






NETWORK
TITLE =S011::STEP-011:EXIT TRANSITION:
    //========================== STEP TRANSFER ===============================//
    // Jump to the common step progression code:                              //
    //------------------------------------------------------------------------//
    JU    COMM;






NETWORK
TITLE =S012: STEP-12::UO_MX_MAKE : Isolate WFI and vessel.
    //================================ STEP HEADER ===========================//
    // STEP012 STEP012 STEP012 STEP012
    // AUTOCODE   AUTOCODE   AUTOCODE   AUTOCODE   AUTOCODE   AUTOCODE   AUTO //
    // STEP012 STEP012 STEP012 STEP012
    //------------------------------------------------------------------------//
    // Log operator confirmation.
    // Isolate WFI and vessel.
    //------------------------------------------------------------------------//
S012: NOP   0;

      SET;
      R     #sqSequencer.STEP.jumpDone[12];
      A     #sqSequencer.CMD.Pause; //If paused jump
      JC    COMM;

NETWORK
TITLE =S012:STEP-12:Begin Action

      A     #sqSequencer.STEP.Finished;
      JC    A012; // Exit Action code, Jump to A012 Transition code

      //----------------------------------------------------------------------//
      // Begin step Action:                                                   //
      //----------------------------------------------------------------------//
      A     #sqSequencer.STEP.Active;
      JC    L012; // Action number loaded, Jump to L012--Step Action List

      //----------------------------------------------------------------------//
      // Load Default/Initial Step action number:                             //
      //----------------------------------------------------------------------//
      S     #sqSequencer.STEP.Active;
      S     #sqStepTimer.IN;
      L     1; //First Action, Step must contain Minimum one action
      T     #sqSequencer.STEP.ActionNumber;

//----------------------------------------------------------------------------//
// Step action list.                                                          //
// aann=mini Action step number(aa) inside main step number(nn)               //
// First Action aa00, Second action ab00, Third ac00, etc.                    //
//----------------------------------------------------------------------------//
L012: NOP   0;

      L     #sqSequencer.STEP.ActionNumber;
      JL    r012; //Wrong Action number
      JU    _012; //Action error handling
       JU    aa12; //ACTION-01
JU    ab12; //ACTION-02
JU    ac12; //ACTION-03


//----------------------------------------------------------------------------//
// More step action in the list can be inserted here, upto ab is tested:      //
//----------------------------------------------------------------------------//
r012: NOP   0; //Wrong action number
      S     #sqSequencer.Error_Fault;
      JU    k012; //Exit
_012: NOP   0; // Action error handling
      JU    k012; // Exit






NETWORK
TITLE =S012:: STEP-012:: : ACTION CODE
    //================================ ACT HEADER ============================//
    // ACTION ACTION ACTION ACTION ACTION ACTION ACTION ACTION ACTION ACTION  //
    // AUTOCODE   AUTOCODE   AUTOCODE   AUTOCODE   AUTOCODE   AUTOCODE   AUTO //
    // ACTION ACTION ACTION ACTION ACTION ACTION ACTION ACTION ACTION ACTION  //
    //------------------------------------------------------------------------//
    // //Reset vessel connection EMs
    aa12: NOP   0;

    //------------------------------------------------------------------------//
    // ACT ACT ACT ACT ACT ACT ACT ACT ACT ACT ACT ACT ACT ACT ACT ACT ACT    //
    //------------------------------------------------------------------------//
    L "dbCONST".BLK.CMD.STOP;
T  #_emc_water_cmd;
T  #_emv_vessel_cmd;

    //------------------------------------------------------------------------//
    // VERIFY  VERIFY VERIFY VERIFY VERIFY VERIFY VERIFY VERIFY VERIFY VERIFY //
    //------------------------------------------------------------------------//
    A(;
L #_emc_water_state;
L "dbCONST".BLK.STATE.STOPPED;
==I;
);
A(;
L #_emv_vessel_state;
L "dbCONST".BLK.STATE.STOPPED;
==I;
);
    S     #sqSequencer.STEP.ActionVerified; //Action verified

    //------------------------------------------------------------------------//
    // Action done:                                                           //
    //------------------------------------------------------------------------//
    O     #sqSequencer.STEP.ActionVerified;
    O     #smc.NO_VERIFIC;       //No verification , bypass verification code
    S     #sqSequencer.STEP.ActionFinished;






    //============================= ACT FOOTER ===============================//
    // AUTOCODE   AUTOCODE   AUTOCODE   AUTOCODE   AUTOCODE   AUTOCODE   AUTO //
    // Get Ready after action finished:                                       //
    //------------------------------------------------------------------------//
    A     #sqSequencer.STEP.ActionFinished;
    JCN   k012;

    //------------------------------------------------------------------------//
    // Reset Action finished flag, ready for next step action:                //
    //------------------------------------------------------------------------//
    R     #sqSequencer.STEP.ActionVerified;
    R     #sqSequencer.STEP.ActionFinished;

    //------------------------------------------------------------------------//
    // Load Next Step Action number:                                          //
    //------------------------------------------------------------------------//
    L     02; //Load next Action
    T     #sqSequencer.STEP.ActionNumber;






NETWORK
TITLE =S012:: STEP-012:: : ACTION CODE
    //================================ ACT HEADER ============================//
    // ACTION ACTION ACTION ACTION ACTION ACTION ACTION ACTION ACTION ACTION  //
    // AUTOCODE   AUTOCODE   AUTOCODE   AUTOCODE   AUTOCODE   AUTOCODE   AUTO //
    // ACTION ACTION ACTION ACTION ACTION ACTION ACTION ACTION ACTION ACTION  //
    //------------------------------------------------------------------------//
    // //Log time when operator confirmed manufacturing complete, start timer and isolate WFI.
    ab12: NOP   0;

    //------------------------------------------------------------------------//
    // ACT ACT ACT ACT ACT ACT ACT ACT ACT ACT ACT ACT ACT ACT ACT ACT ACT    //
    //------------------------------------------------------------------------//
    //Log time when operator confirmed manufacturing complete.
SET;
S #_log_msg_pmo_complete;
R #_prompt_pmo_confirm_yes;
R #_make_active;
// Isolate WFI
L "dbCONST".BLK.EMC2.SUBS.ISOLATE;
T #_emc_water_subs;
L "dbCONST".BLK.CMD.START;
T #_emc_water_cmd;

    //------------------------------------------------------------------------//
    // VERIFY  VERIFY VERIFY VERIFY VERIFY VERIFY VERIFY VERIFY VERIFY VERIFY //
    //------------------------------------------------------------------------//
    //Verify if emc_water changed to substate ISOLATE.
A(;
L #_emc_water_subs;
L "dbCONST".BLK.EMC2.SUBS.ISOLATE;
==I;
);
    S     #sqSequencer.STEP.ActionVerified; //Action verified

    //------------------------------------------------------------------------//
    // Action done:                                                           //
    //------------------------------------------------------------------------//
    O     #sqSequencer.STEP.ActionVerified;
    O     #smc.NO_VERIFIC;       //No verification , bypass verification code
    S     #sqSequencer.STEP.ActionFinished;






    //============================= ACT FOOTER ===============================//
    // AUTOCODE   AUTOCODE   AUTOCODE   AUTOCODE   AUTOCODE   AUTOCODE   AUTO //
    // Get Ready after action finished:                                       //
    //------------------------------------------------------------------------//
    A     #sqSequencer.STEP.ActionFinished;
    JCN   k012;

    //------------------------------------------------------------------------//
    // Reset Action finished flag, ready for next step action:                //
    //------------------------------------------------------------------------//
    R     #sqSequencer.STEP.ActionVerified;
    R     #sqSequencer.STEP.ActionFinished;

    //------------------------------------------------------------------------//
    // Load Next Step Action number:                                          //
    //------------------------------------------------------------------------//
    L     03; //Load next Action
    T     #sqSequencer.STEP.ActionNumber;






NETWORK
TITLE =S012:: STEP-012:: : ACTION CODE
    //================================ ACT HEADER ============================//
    // ACTION ACTION ACTION ACTION ACTION ACTION ACTION ACTION ACTION ACTION  //
    // AUTOCODE   AUTOCODE   AUTOCODE   AUTOCODE   AUTOCODE   AUTOCODE   AUTO //
    // ACTION ACTION ACTION ACTION ACTION ACTION ACTION ACTION ACTION ACTION  //
    //------------------------------------------------------------------------//
    // //Isolate Vessel
    ac12: NOP   0;

    //------------------------------------------------------------------------//
    // ACT ACT ACT ACT ACT ACT ACT ACT ACT ACT ACT ACT ACT ACT ACT ACT ACT    //
    //------------------------------------------------------------------------//
    // Isolate Vessel
L     "dbCONST".BLK.EMV1.SUBS.ISOLATE;
T     #_emv_vessel_subs;
L     "dbCONST".BLK.CMD.START;
T     #_emv_vessel_cmd;

    //------------------------------------------------------------------------//
    // VERIFY  VERIFY VERIFY VERIFY VERIFY VERIFY VERIFY VERIFY VERIFY VERIFY //
    //------------------------------------------------------------------------//
    A(;
L     #_emv_vessel_subs;
L     "dbCONST".BLK.EMV1.SUBS.ISOLATE;
==I;
);
    S     #sqSequencer.STEP.ActionVerified; //Action verified

    //------------------------------------------------------------------------//
    // Action done:                                                           //
    //------------------------------------------------------------------------//
    O     #sqSequencer.STEP.ActionVerified;
    O     #smc.NO_VERIFIC;       //No verification , bypass verification code
    S     #sqSequencer.STEP.ActionFinished;






    //============================= STEP FOOTER ==============================//
    // AUTOCODE   AUTOCODE   AUTOCODE   AUTOCODE   AUTOCODE   AUTOCODE   AUTO //
    // Get Ready after action finished:                                       //
    //------------------------------------------------------------------------//
    A     #sqSequencer.STEP.ActionFinished;
    JCN   k012;

    //------------------------------------------------------------------------//
    // Reset Action finished flag, ready for next step action:                //
    //------------------------------------------------------------------------//
    R     #sqSequencer.STEP.ActionVerified;
    R     #sqSequencer.STEP.ActionFinished;

    //------------------------------------------------------------------------//
    // If ALL actions are finished:                                           //
    //------------------------------------------------------------------------//
    SET   ;
    S     #sqSequencer.STEP.Finished;
    R     #sqSequencer.STEP.Active;
    S     #sqSequencer.STEP.Done[12];

    //------------------------------------------------------------------------//
    // End Step action(s):                                                    //
    //------------------------------------------------------------------------//
    JU    k012;

//----------------------------------------------------------------------------//
// Finished Step Action(s):                                                   //
//----------------------------------------------------------------------------//
k012: NOP   0;

    A     #sqStepTimerExpired;
    S     #sqSequencer.STEP.WithError[12]; // Step error flag
    S     #sqSequencer.Error_Fault;
    R     #sqStepTimer.IN;

NETWORK
TITLE =S012:STEP-012::Begin Transition
    //------------------------------------------------------------------------//
    // Begin the transition code:                                             //
    //------------------------------------------------------------------------//
    A012: NOP   0;
    R     #sqStepTimer.IN;






    //============================= TRAN HEADER ==============================//
    // AUTOCODE   AUTOCODE   AUTOCODE   AUTOCODE   AUTOCODE   AUTOCODE   AUTO //
    // Bypass transition if manual jump:                                      //
    //------------------------------------------------------------------------//
    A     #sqSequencer.STEP.Finished;
    A     #smc.TRN_AND_JUMP;     //Manual jump is set Transition as bypassed
    JCN   COMM;              //exit

NETWORK
TITLE =S012::STEP 012:TRAN 016: WFI and Vessel isolated?
//----------------------------------------------------------------------------//
// TRAN   TRAN   TRAN   TRAN   TRAN   TRAN   TRAN   TRAN   TRAN   TRAN   TRAN //
// TRAN   TRAN   TRAN   TRAN   TRAN   TRAN   TRAN   TRAN   TRAN   TRAN   TRAN //
//----------------------------------------------------------------------------//
// WFI and Vessel isolated.
//----------------------------------------------------------------------------//
// CONDITION   CONDITION   CONDITION   CONDITION   CONDITION   CONDITION   CO //
// CONDITION   CONDITION   CONDITION   CONDITION   CONDITION   CONDITION   CO //
//----------------------------------------------------------------------------//
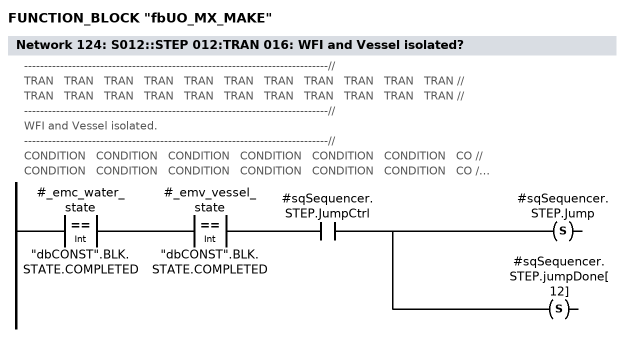
A(;
L     #_emc_water_state;
L   "dbCONST".BLK.STATE.COMPLETED;
==I;
);
A(;
L    #_emv_vessel_state;
L   "dbCONST".BLK.STATE.COMPLETED;
==I;
);






    //============================= TRAN FOOTER ==============================//
    // Transition jump control:                                               //
    //------------------------------------------------------------------------//
    A     #sqSequencer.STEP.JumpCtrl;
    S     #sqSequencer.STEP.Jump;
    S     #sqSequencer.STEP.jumpDone[12];

NETWORK
TITLE =S012:t016::TRANS-v: EXIT TRANSITION AND READY THE NEXT STEP
    //------------------------------------------------------------------------//
    // Check the jump flag and jump to the next step if the transition        //
    // condition is true and has set the jump flag:                           //
    //------------------------------------------------------------------------//
    A     #sqSequencer.STEP.Jump;
    JCN   x016;

    R     #sqSequencer.STEP.Jump;
    R     #sqSequencer.STEP.Finished;

    L     13;     // Load next STEPNO to jump to if transition satisfied
    T     #sqSequencer.STEP.NumberNext; //Next Step13.

    JU    COMM;              // Transition satisfied, Exit, go to next step
x016: NOP   0;






NETWORK
TITLE =S012::STEP-012:EXIT TRANSITION:
    //========================== STEP TRANSFER ===============================//
    // Jump to the common step progression code:                              //
    //------------------------------------------------------------------------//
    JU    COMM;






NETWORK
TITLE =S013: STEP-13::UO_MX_MAKE : Manufacturing Unit Operation Completed
    //================================ STEP HEADER ===========================//
    // STEP013 STEP013 STEP013 STEP013
    // AUTOCODE   AUTOCODE   AUTOCODE   AUTOCODE   AUTOCODE   AUTOCODE   AUTO //
    // STEP013 STEP013 STEP013 STEP013
    //------------------------------------------------------------------------//
    // Set all devices to safe state.
    // Enable LPCA pressure control and enable Mx Manway alarm.
    // Enable Mx Low and LowLow Pressure Alarm.
    // Set other equipment to safe state.
    // Log Mx Make operation end time.
    //------------------------------------------------------------------------//
S013: NOP   0;

      SET;
      R     #sqSequencer.STEP.jumpDone[13];
      A     #sqSequencer.CMD.Pause; //If paused jump
      JC    COMM;

NETWORK
TITLE =S013:STEP-13:Begin Action

      A     #sqSequencer.STEP.Finished;
      JC    A013; // Exit Action code, Jump to A013 Transition code

      //----------------------------------------------------------------------//
      // Begin step Action:                                                   //
      //----------------------------------------------------------------------//
      A     #sqSequencer.STEP.Active;
      JC    L013; // Action number loaded, Jump to L013--Step Action List

      //----------------------------------------------------------------------//
      // Load Default/Initial Step action number:                             //
      //----------------------------------------------------------------------//
      S     #sqSequencer.STEP.Active;
      S     #sqStepTimer.IN;
      L     1; //First Action, Step must contain Minimum one action
      T     #sqSequencer.STEP.ActionNumber;

//----------------------------------------------------------------------------//
// Step action list.                                                          //
// aann=mini Action step number(aa) inside main step number(nn)               //
// First Action aa00, Second action ab00, Third ac00, etc.                    //
//----------------------------------------------------------------------------//
L013: NOP   0;

      L     #sqSequencer.STEP.ActionNumber;
      JL    r013; //Wrong Action number
      JU    _013; //Action error handling
       JU    aa13; //ACTION-01
JU    ab13; //ACTION-02


//----------------------------------------------------------------------------//
// More step action in the list can be inserted here, upto ab is tested:      //
//----------------------------------------------------------------------------//
r013: NOP   0; //Wrong action number
      S     #sqSequencer.Error_Fault;
      JU    k013; //Exit
_013: NOP   0; // Action error handling
      JU    k013; // Exit






NETWORK
TITLE =S013:: STEP-013:: : ACTION CODE
    //================================ ACT HEADER ============================//
    // ACTION ACTION ACTION ACTION ACTION ACTION ACTION ACTION ACTION ACTION  //
    // AUTOCODE   AUTOCODE   AUTOCODE   AUTOCODE   AUTOCODE   AUTOCODE   AUTO //
    // ACTION ACTION ACTION ACTION ACTION ACTION ACTION ACTION ACTION ACTION  //
    //------------------------------------------------------------------------//
    // //Enable LPCA pressure control and enable Mx Manway alarm.
    aa13: NOP   0;

    //------------------------------------------------------------------------//
    // ACT ACT ACT ACT ACT ACT ACT ACT ACT ACT ACT ACT ACT ACT ACT ACT ACT    //
    //------------------------------------------------------------------------//
    //Stop emv_vessel.
L "dbCONST".BLK.CMD.STOP;
T #_emv_vessel_cmd;
T #_emv_inlet_cmd;
T #_emm_vessel_cmd;
T  #_ema_vessel_cmd;
T  #_emc_gas_cmd;
T  #_emc_water_cmd;

    //------------------------------------------------------------------------//
    // VERIFY  VERIFY VERIFY VERIFY VERIFY VERIFY VERIFY VERIFY VERIFY VERIFY //
    //------------------------------------------------------------------------//
    //Verify emv_vessel stopped.
A(;
L #_emv_vessel_state;
L "dbCONST".BLK.STATE.STOPPED;
==I;
);
    S     #sqSequencer.STEP.ActionVerified; //Action verified

    //------------------------------------------------------------------------//
    // Action done:                                                           //
    //------------------------------------------------------------------------//
    O     #sqSequencer.STEP.ActionVerified;
    O     #smc.NO_VERIFIC;       //No verification , bypass verification code
    S     #sqSequencer.STEP.ActionFinished;






    //============================= ACT FOOTER ===============================//
    // AUTOCODE   AUTOCODE   AUTOCODE   AUTOCODE   AUTOCODE   AUTOCODE   AUTO //
    // Get Ready after action finished:                                       //
    //------------------------------------------------------------------------//
    A     #sqSequencer.STEP.ActionFinished;
    JCN   k013;

    //------------------------------------------------------------------------//
    // Reset Action finished flag, ready for next step action:                //
    //------------------------------------------------------------------------//
    R     #sqSequencer.STEP.ActionVerified;
    R     #sqSequencer.STEP.ActionFinished;

    //------------------------------------------------------------------------//
    // Load Next Step Action number:                                          //
    //------------------------------------------------------------------------//
    L     02; //Load next Action
    T     #sqSequencer.STEP.ActionNumber;






NETWORK
TITLE =S013:: STEP-013:: : ACTION CODE
    //================================ ACT HEADER ============================//
    // ACTION ACTION ACTION ACTION ACTION ACTION ACTION ACTION ACTION ACTION  //
    // AUTOCODE   AUTOCODE   AUTOCODE   AUTOCODE   AUTOCODE   AUTOCODE   AUTO //
    // ACTION ACTION ACTION ACTION ACTION ACTION ACTION ACTION ACTION ACTION  //
    //------------------------------------------------------------------------//
    // //Set other equipment to safe state and reset flags.
    // //Log Mx Make operation end time.
    ab13: NOP   0;

    //------------------------------------------------------------------------//
    // ACT ACT ACT ACT ACT ACT ACT ACT ACT ACT ACT ACT ACT ACT ACT ACT ACT    //
    //------------------------------------------------------------------------//
    //Set substate to safe state and stop equipments..
L "dbCONST".BLK.CMD.STOP;
T  #_emc_water_cmd;
T  #_ema_vessel_cmd;
T  #_emv_vessel_cmd;
T #_emv_inlet_cmd;
T  #_emm_vessel_cmd;
T #_emv_inlet_cmd;

//Reset flags.
R #_cmd_measure;
R #_cmd_charge;
R #_cmd_mix;
R #_cmd_manway;
R #_cmd_complete;

//Log MAKE operation end time.
SET;
S #_log_msg_make_end;

    //------------------------------------------------------------------------//
    // VERIFY  VERIFY VERIFY VERIFY VERIFY VERIFY VERIFY VERIFY VERIFY VERIFY //
    //------------------------------------------------------------------------//
    A(;
L #_emc_water_state;
L "dbCONST".BLK.STATE.STOPPED;
==I;
);
A(;
L #_ema_vessel_state;
L "dbCONST".BLK.STATE.STOPPED;
==I;
);
A(;
L #_emv_vessel_state;
L "dbCONST".BLK.STATE.STOPPED;
==I;
);
A(;
L #_emm_vessel_state;
L "dbCONST".BLK.STATE.STOPPED;
==I;
);
    S     #sqSequencer.STEP.ActionVerified; //Action verified

    //------------------------------------------------------------------------//
    // Action done:                                                           //
    //------------------------------------------------------------------------//
    O     #sqSequencer.STEP.ActionVerified;
    O     #smc.NO_VERIFIC;       //No verification , bypass verification code
    S     #sqSequencer.STEP.ActionFinished;






    //============================= STEP FOOTER ==============================//
    // AUTOCODE   AUTOCODE   AUTOCODE   AUTOCODE   AUTOCODE   AUTOCODE   AUTO //
    // Get Ready after action finished:                                       //
    //------------------------------------------------------------------------//
    A     #sqSequencer.STEP.ActionFinished;
    JCN   k013;

    //------------------------------------------------------------------------//
    // Reset Action finished flag, ready for next step action:                //
    //------------------------------------------------------------------------//
    R     #sqSequencer.STEP.ActionVerified;
    R     #sqSequencer.STEP.ActionFinished;

    //------------------------------------------------------------------------//
    // If ALL actions are finished:                                           //
    //------------------------------------------------------------------------//
    SET   ;
    S     #sqSequencer.STEP.Finished;
    R     #sqSequencer.STEP.Active;
    S     #sqSequencer.STEP.Done[13];

    //------------------------------------------------------------------------//
    // End Step action(s):                                                    //
    //------------------------------------------------------------------------//
    JU    k013;

//----------------------------------------------------------------------------//
// Finished Step Action(s):                                                   //
//----------------------------------------------------------------------------//
k013: NOP   0;

    A     #sqStepTimerExpired;
    S     #sqSequencer.STEP.WithError[13]; // Step error flag
    S     #sqSequencer.Error_Fault;
    R     #sqStepTimer.IN;

NETWORK
TITLE =S013:STEP-013::Begin Transition
    //------------------------------------------------------------------------//
    // Begin the transition code:                                             //
    //------------------------------------------------------------------------//
    A013: NOP   0;
    R     #sqStepTimer.IN;






NETWORK
TITLE =S013::STEP-013:EXIT TRANSITION:
    //========================== STEP TRANSFER ===============================//
    // Jump to the common step progression code:                              //
    //------------------------------------------------------------------------//
    JU    COMM;






NETWORK
TITLE =Sequencer Common Code, Execute in Each Scan
    //============================ SEQ FOOTER ================================//
    // AUTOCODE   AUTOCODE   AUTOCODE   AUTOCODE   AUTOCODE   AUTOCODE   AUTO //
    // Common code to execute each scan:                                      //
    //------------------------------------------------------------------------//
    COMM: NOP   0;

NETWORK
TITLE =Retentive/Non Retentive Selectable Run timer
    CALL #sqRunTimer (
        TIME_H               := #sqRunTimer.TIME_H,
        TIME_M               := #sqRunTimer.TIME_M,
        TIME_S               := #sqRunTimer.TIME_S,
        ENABLE               := #sqRunTimer.ENABLE,
        RESET                := #sqRunTimer.RESET,
        PAUSE                := #sqRunTimer.PAUSE,
        NON_RET              := #sqRunTimer.NON_RET,
        RMNG_H               := #sqRunTimer.RMNG_H,
        RMNG_M               := #sqRunTimer.RMNG_M,
        RMNG_S               := #sqRunTimer.RMNG_S,
        TIME_EXPIRED         := #sqRunTimer.TIME_EXPIRED,
        TMR_RUNNG            := #sqRunTimer.TMR_RUNNG
    );

NETWORK
TITLE =Sequencer Step Timer
    CALL #sqStepTimer (
        IN                   := #sqStepTimer.IN,
        PT                   := "dbCONST".SEQ.STEP_TIME,
        Q                    := #sqStepTimerExpired,
        ET                   := #sqStepTimerElapsed
    );

NETWORK
TITLE =Sequencer Timer
    CALL #SQ_TIMER (
        IN                   := #sqSeqTimerStart,
        PT                   := #SQ_TIMER.PT,
        Q                    := #sqSeqTimerExpired,
        ET                   := #sqSeqTimerElapsed
    );

    CALL #SQ_TIMER2 (
        IN                   := #sqSeqTimerStart2,
        PT                   := #SQ_TIMER2.PT,
        Q                    := #sqSeqTimerExpired2,
        ET                   := #sqSeqTimerElapsed2
    );

NETWORK
TITLE =Sequencer Timer
    CALL #SQ_TIMER3 (
        IN                   := #sqSeqTimerStart3,
        PT                   := #SQ_TIMER3.PT,
        Q                    := #sqSeqTimerExpired3,
        ET                   := #sqSeqTimerElapsed3
    );

NETWORK
TITLE =General Assignments

    L     #sqSequencer.STEP.NumberNext;
    T     #smc.NXT_STEP;
    T     #sqSequencer.STEP.NumberCurrent;
    T     #smc.CURSTEP;

    A     #sqSequencer.STEP.Active;
    =     #smc.S_ACTIVE;

    A     #sqSequencer.Error_Fault;
    =     #smc.ERR_FAULT;

NETWORK
TITLE = Stop command completion
    A    #smc.OFF_IDLE;
    A    #sqSequencer.STEP.Done[13];
    AN   #sqSequencer.STEP.WithError[13];
    JCN NotStopCmd;
    R    #smc.PAUSED;
    R    #sqSequencer.STEP.Error_Fault;
    R    #sqSequencer.Error_Fault;
    L    "dbCONST".SEQ.STATE.OFF_IDLE;
    T    #smc.SQ_STATE;
NotStopCmd:   NOP 0;

    A    #smc.OFF_IDLE;
    AN    #sqSequencer.STEP.Done[13];
    AN    #sqSequencer.STEP.WithError[13];
    JCN   _stopAction;
    R     #sqSequencer.STEP.Finished;
    R     #smc.PAUSED;
    R     #sqSequencer.STEP.Error_Fault;
    R     #sqSequencer.Error_Fault;
_stopAction:   NOP 0;

NETWORK
TITLE =Sequencer Finished

    AN    #smc.OFF_IDLE;
    AN    #smc.PAUSED;
    A     #sqSequencer.STEP.Done[13];
    =     #sqSequencer.Finished;
    =     #smc.SQ_FINISHED;
    JCN   fnsd;
    L     "dbCONST".SEQ.STATE.COMPLETED;
    T     #smc.SQ_STATE;
    R     #smc.PAUSED;
    R     #sqSequencer.STEP.Error_Fault;
    R     #sqSequencer.Error_Fault;
fnsd: NOP   0;

    //------------------------------------------------------------------------//
    // Reset Finished flag if SQ OFF for Last step to scan:                   //
    //------------------------------------------------------------------------//
    A     #smc.ABORTED;
    AN    #sqSequencer.STEP.Done[13];
    AN    #sqSequencer.STEP.WithError[13];
    JCN   _abrt_end;
    R     #sqSequencer.STEP.Finished;
    R     #smc.PAUSED;
    R     #sqSequencer.STEP.Error_Fault;
    R     #sqSequencer.Error_Fault;
    L     "dbCONST".SEQ.STATE.ABORTED;
    T     #smc.SQ_STATE;
_abrt_end: NOP   0;

    //------------------------------------------------------------------------//
    // Visio Common Code Begin:                                               //
    //------------------------------------------------------------------------//


//----------------------------------------------------------------------------//
// End of Sequencer:                                                          //
//----------------------------------------------------------------------------//
END_FUNCTION_BLOCK

